FUNCTION_BLOCK FB_Foerderband
VAR_INPUT
	//Steuereingänge
	benable : BOOL;
	bexecute : BOOL;
	bhalt : BOOL;
	rVel : INT := 30; //mm per s
	
	eDirection : MC_Direction := MC_Positive_Direction;
END_VAR
VAR_OUTPUT
	estate: eBetriebszustand;
END_VAR
VAR
	nstate : INT := 0;
	
	//Motion Blöcke der Tc2_Mc2
	mcReset : MC_Reset;
	mcPower : MC_Power;
	mcMove : MC_MoveVelocity;
	mcHalt : MC_Halt;
	
	bAxPower : BOOL;
	bAXMove : BOOL;
	
	fbTon	:Ton;
END_VAR
VAR_IN_OUT
	ax : AXIS_REF;
END_VAR

// update our axis
ax.ReadStatus();

mcReset(Axis := ax); 

mcPower(
	Axis:= ax, 
	Enable:= bAxPower, 
	Enable_Positive:= bAxPower, 
	Enable_Negative:= bAxPower, 
	Override:= 100);

mcMove(
	Axis:= ax, 
	Execute:= bAxMove , 
	Velocity:= rVel,
	Acceleration:= 60.0, 
	Direction:= eDirection);
	
mcHalt(
	Axis:= ax, 
	Execute:= ,
	Deceleration:= 60.0);
	
fbTon(
  IN := bhalt,   
  PT := T#1S
);
	

IF NOT benable THEN
	nstate := 0;
END_IF

CASE nstate OF 
	
	0: //off
	estate := eBetriebszustand.off;
	bAxPower := FALSE;
	bAxMove := FALSE;
	
	IF McPower.Status AND benable THEN
		nstate := 20; //Ready
	END_IF
	IF NOT McPower.Status AND bEnable THEN
		nstate:=10;
	END_IF
	
	10: // INIT_Reset
	estate := eBetriebszustand.init;
	mcReset.Execute := TRUE;
	bAxPower:= FALSE;
	bAxMove:= FALSE;
	bhalt:= False;
	
	IF McReset.Done THEN
		nstate:= 11; //INIT-Power
	END_IF
	
	11: //INIT-Power
	estate := eBetriebszustand.init;
	bAxPower := TRUE;
	
	IF Mcpower.Status THEN
		nstate := 20; //Ready
	END_IF
	
	20: //Ready
	estate:= eBetriebszustand.ready;
	mcHalt.Execute := FALSE;
	bAxMove := FALSE;
	
	IF bexecute THEN
		nstate := 30; // Move
	END_IF
	
	30: //Move
	estate := eBetriebszustand.production;
	bAxMove := TRUE;

	IF bhalt THEN
		nstate := 31; //Warten
	END_IF
	
	31: //Warten
	estate := eBetriebszustand.production;
	bAxMove := TRUE;
	
	IF fbTOn.Q THEN
		nstate:= 32; //Halten
	END_IF
	
	32: //Halten
	estate := eBetriebszustand.production;
    mcHalt.Execute := TRUE;
	
	
	IF NOT bexecute THEN
		nstate := 20; // Ready
	END_IF
	
END_CASE

END_FUNCTION_BLOCK

(* stored: Version 1.1.0.1, ProductVersion 3.1.4024.15
   POU FB_Foerderband: Id {1c512206-a637-4e93-9a74-064188af753d}, SpecialFunc None *)
